// TIA Portal V20 export
TYPE "type_emRelations_em2_cmStatus"
// stored: Access Published, Namespace Unit1
   STRUCT
      cmSuctionPadTopUpDown { S7_SetPoint := 'True'} : "LBC_typeTwoWayActuatorControlNode";
      cmSuctionPadBtmUpDown { ExternalAccessible := 'False'; ExternalVisible := 'False'; ExternalWritable := 'False'} : "LBC_typeTwoWayActuatorControlNode";
      cmCutterUpDown { ExternalWritable := 'False'} : "LBC_typeTwoWayActuatorControlNode";
      cmTapeTopUpDown { ExternalAccessible := 'False'; ExternalVisible := 'False'; ExternalWritable := 'False'; S7_SetPoint := 'True'} : "LBC_typeTwoWayActuatorControlNode";
      cmTapeBtmUpDown { ExternalAccessible := 'False'; ExternalVisible := 'False'; ExternalWritable := 'False'; S7_SetPoint := 'True'} : "LBC_typeTwoWayActuatorControlNode";
      cmSpliceHeadRotateTopFwdBwd { ExternalAccessible := 'False'; ExternalVisible := 'False'; ExternalWritable := 'False'} : "LBC_typeTwoWayActuatorControlNode";
      cmSpliceHeadRotateBtmFwdBwd { S7_SetPoint := 'True'} : "LBC_typeTwoWayActuatorControlNode";
      cmSuctionPadTopLeftVaccum { S7_SetPoint := 'True'} : "LBC_typeTwoWayActuatorControlNode";
      cmSuctionPadTopRightVaccum { S7_SetPoint := 'True'} : "LBC_typeTwoWayActuatorControlNode";
      cmSuctionPadBtmLeftVaccum { S7_SetPoint := 'True'} : "LBC_typeTwoWayActuatorControlNode";
      cmSuctionPadBtmRightVaccum { S7_SetPoint := 'True'} : "LBC_typeTwoWayActuatorControlNode";
      cmSuctionPadTopTapeVaccum { S7_SetPoint := 'True'} : "LBC_typeTwoWayActuatorControlNode";
      cmSuctionPadBtmTapeVaccum { S7_SetPoint := 'True'} : "LBC_typeTwoWayActuatorControlNode";
   END_STRUCT;
END_TYPE
